SUBAPPLICATION RegisterServicePartialOpcUa (* Register a Service using OPC UA. The system information is encapsulated *)
  (* Standard: 61499-2; Description: Copyright (c) 2019 fortiss GmbH This program and the accompanying materials are made available under the terms of the Eclipse Public License 2.0 which is available at https://www.eclipse.org/legal/epl-2.0/ SPDX-License-Identifier: EPL-2.0 *)
  (* Version 1.0, 2019-09-17, Jose Cabral, fortiss GmbH *)
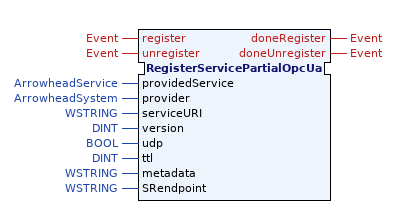
  EVENT_INPUT
    register; (* Register the service *)
    unregister; (* Unregister the service *)
  END_EVENT
  EVENT_OUTPUT
    doneRegister; (* Register finished *)
    doneUnregister; (* Unregister finished *)
  END_EVENT
  VAR_INPUT
    providedService : ArrowheadService; (* The Arrowhead Service object that is provided (SD and supported IDD-s) *)
    provider : ArrowheadSystem; (* ArrowheadSystem that is providing the Service *)
    serviceURI : WSTRING; (* The URL subpath of the Service within the address:port of the Provider *)
    version : DINT; (* The version numbering of the Service provided *)
    udp : BOOL; (* True, if the service is provided via UDP. By default, it is false *)
    ttl : DINT; (* Service validity time period expressed in seconds. This gets converted to a date-time, and stored in the database *)
    metadata : WSTRING; (* Metadata belonging to a service/provider pair *)
    SRendpoint : WSTRING; (* Endpoint (IP:PORT/URI) of the Service Registry *)
  END_VAR
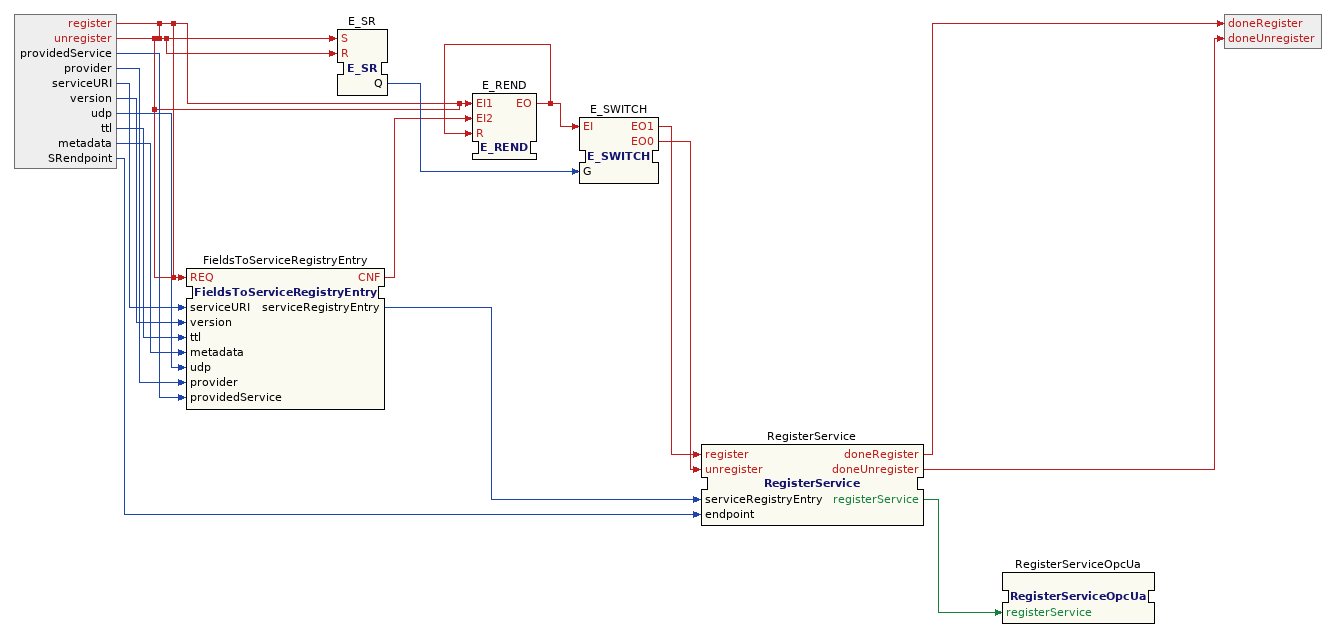
  FBS
    FieldsToServiceRegistryEntry : FieldsToServiceRegistryEntry;
    RegisterService : RegisterService;
    E_SR : E_SR;
    E_SWITCH : E_SWITCH;
    E_REND : E_REND;
    RegisterServiceOpcUa : RegisterServiceOpcUa;
  END_FBS
  EVENT_CONNECTIONS
    RegisterService.doneRegister TO doneRegister;
    RegisterService.doneUnregister TO doneUnregister;
    E_SWITCH.EO1 TO RegisterService.register;
    E_SWITCH.EO0 TO RegisterService.unregister;
    register TO E_SR.S;
    unregister TO E_SR.R;
    register TO FieldsToServiceRegistryEntry.REQ;
    unregister TO FieldsToServiceRegistryEntry.REQ;
    register TO E_REND.EI1;
    unregister TO E_REND.EI1;
    FieldsToServiceRegistryEntry.CNF TO E_REND.EI2;
    E_REND.EO TO E_SWITCH.EI;
    E_REND.EO TO E_REND.R;
  END_CONNECTIONS
  DATA_CONNECTIONS
    FieldsToServiceRegistryEntry.serviceRegistryEntry TO RegisterService.serviceRegistryEntry;
    serviceURI TO FieldsToServiceRegistryEntry.serviceURI;
    version TO FieldsToServiceRegistryEntry.version;
    ttl TO FieldsToServiceRegistryEntry.ttl;
    metadata TO FieldsToServiceRegistryEntry.metadata;
    SRendpoint TO RegisterService.endpoint;
    E_SR.Q TO E_SWITCH.G;
    udp TO FieldsToServiceRegistryEntry.udp;
    provider TO FieldsToServiceRegistryEntry.provider;
    providedService TO FieldsToServiceRegistryEntry.providedService;
  END_CONNECTIONS
  ADAPTER_CONNECTIONS
    RegisterService.registerService TO RegisterServiceOpcUa.registerService;
  END_CONNECTIONS
END_SUBAPPLICATION
